INTERFACE I_Sequence EXTENDS I_Object

METHOD PUBLIC M_Await : BOOL
VAR_INPUT
	sMessage:				STRING(255);
	nID:					ULINT;
	tTimeout:				TIME;
	tDelay:					TIME;	
	bPause:					BOOL;
	bReturn:				BOOL;
	nNumber:				INT;
END_VAR
END_METHOD

METHOD PUBLIC M_Reset : BOOL
VAR_INPUT
END_VAR
END_METHOD

METHOD PUBLIC M_Set : BOOL
VAR_INPUT
	sMessage:				STRING(255);	
	nNumber:				INT;
END_VAR
END_METHOD


PROPERTY PUBLIC P_Number : INT
GET
END_GET
END_PROPERTY

PROPERTY PUBLIC P_Timeout : Bool
GET
END_GET
END_PROPERTY

END_INTERFACE

(* stored: Version 1.1.0.1
   Itf I_Sequence: Id {ab5e2af8-509e-42fb-9956-7609633302ce}
   Method M_Await: Id {02f2d100-ec87-06db-3782-6cf3157df90e}
   Method M_Reset: Id {e251ab4f-9396-0401-239c-77e0cb01bba3}
   Method M_Set: Id {afbddb29-0f1f-0aa2-3bbb-96cf1969180d}
   Property P_Number: Id {631a24ea-a4e3-0d29-2b7c-383d8bcd6e7f}
   Get Get: Id {b1cbf18b-3abe-0f1f-0c64-012ccffcae4c}
   Property P_Timeout: Id {96204bf6-b0ef-0952-2be4-8d90d7b4d741}
   Get Get: Id {ccee302f-09c9-0f54-187e-24621df9bc60} *)
